// TIA Portal project "station 1 complete twin" (V17)

(* hardware
DEVICE "S7-1500/ET200MP station_1"  S7-1500 station
   slot 0: "Rail_0"  Rack  6ES7 590-1***0-0AA0
   slot 1: "PLC_1"  CPU 1511C-1 PN  6ES7 511-1CK01-0AB0  V2.6
      slot 3: "CPU display_1"  6ES7591-1AA00-0AA0
      slot 32768: "PROFINET interface_1"  X1
         slot 32769: "Port_1"  X1 P1
         slot 32770: "Port_2"  X1 P2
*)

// ===== PLC "PLC_1"  CPU 1511C-1 PN =====

VAR_GLOBAL   // PLC tag table "Default tag table"
   "Tag_1" AT %M0.0 : Bool;
END_VAR

DATA_BLOCK "Station 1"   // DB1
{ S7_Optimized_Access := 'TRUE' }
VERSION : 0.1
   VAR
      Start : Bool;
      Stop : Bool;
      Feed_cylinder : Bool;
      Carriage : Bool;
      Pick_Up_Cylinder : Bool;
      Gripper : Bool;
      System_ON : Bool;
      Workpiece_present : Bool;
      Steps : Int;
      Feed_Cyl_Fully_Extended : Bool;
      Feed_Cyl_Fully_Retracted : Bool;
      Gripper_fully_extended : Bool;
      Gripper_fully_retracted : Bool;
      Carriage_fully_extended : Bool;
      Carriage_fully_retracted : Bool;
   END_VAR
BEGIN
END_DATA_BLOCK

ORGANIZATION_BLOCK "Main"   // OB1, LAD, ProgramCycle
TITLE = "Main Program Sweep (Cycle)"
{ S7_Optimized_Access := 'TRUE' }
VERSION : 0.1
   VAR_INPUT
      Initial_Call : Bool;   // Initial call of this OB
      Remanence : Bool;   // =True, if remanent data are available
   END_VAR
   VAR_TEMP   // added for the SCL form of the ladder/FBD networks
      _w1 : Bool;
   END_VAR
BEGIN

REGION Network 1: Pressing the start button
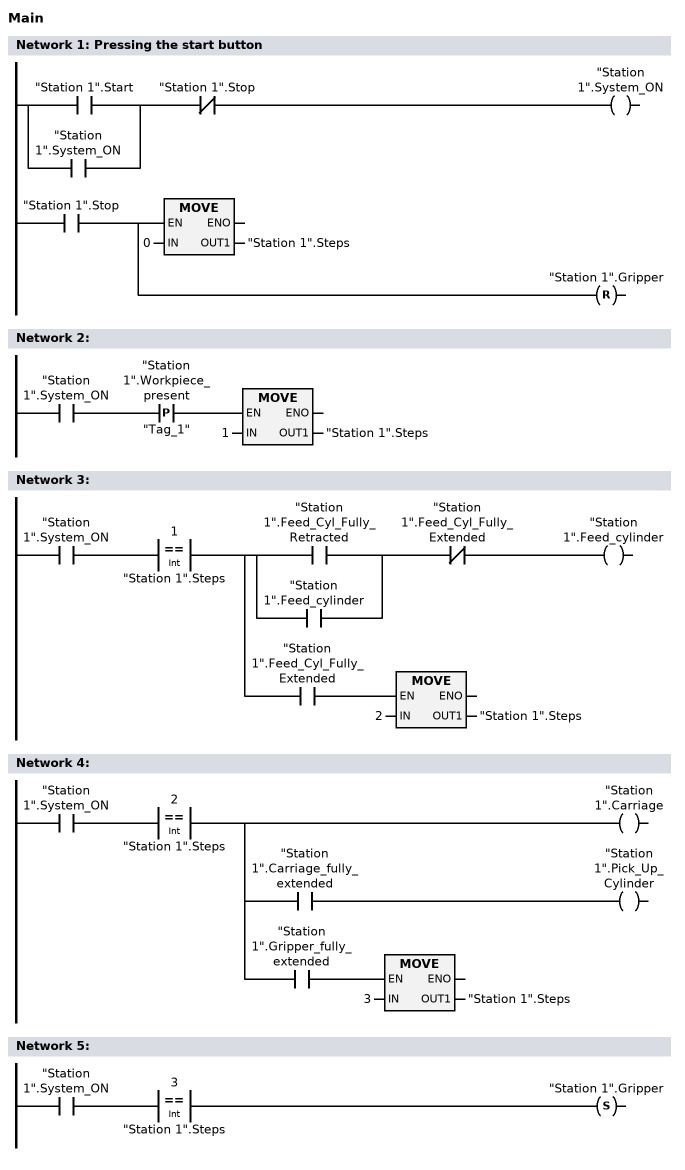
   RUNG wire#powerrail
      Contact( "Station 1".Start )
      wire#w1
      I_Contact( "Station 1".Stop )
      Coil( "Station 1".System_ON )
   END_RUNG
   RUNG wire#powerrail
      Contact( "Station 1".System_ON )
   END_RUNG wire#w1
   RUNG wire#powerrail
      Contact( "Station 1".Stop )
      wire#w2
      Move(in := 0, out1 => "Station 1".Steps)
   END_RUNG
   RUNG wire#w2
      R_Coil( "Station 1".Gripper )
   END_RUNG
   // the same network as SCL:
   "Station 1".System_ON := ("Station 1".Start OR "Station 1".System_ON) AND NOT "Station 1".Stop;
   IF "Station 1".Stop THEN
       "Station 1".Steps := 0;
       "Station 1".Gripper := FALSE;
   END_IF;
END_REGION

REGION Network 2
   RUNG wire#powerrail
      Contact( "Station 1".System_ON )
      P_Contact(operand := "Station 1".Workpiece_present, bit := "Tag_1")
      Move(in := 1, out1 => "Station 1".Steps)
   END_RUNG
   // the same network as SCL:
   #_w1 := "Station 1".System_ON AND "Station 1".Workpiece_present AND NOT "Tag_1";   // rising edge of "Station 1".Workpiece_present
   "Tag_1" := "Station 1".Workpiece_present;
   IF #_w1 THEN "Station 1".Steps := 1; END_IF;
END_REGION

REGION Network 3
   RUNG wire#powerrail
      Contact( "Station 1".System_ON )
      { S7_Templates := "SrcType := Int" } EQ_Contact(in1 := 1, in2 := "Station 1".Steps)
      wire#w1
      Contact( "Station 1".Feed_Cyl_Fully_Retracted )
      wire#w2
      I_Contact( "Station 1".Feed_Cyl_Fully_Extended )
      Coil( "Station 1".Feed_cylinder )
   END_RUNG
   RUNG wire#w1
      Contact( "Station 1".Feed_cylinder )
   END_RUNG wire#w2
   RUNG wire#w1
      Contact( "Station 1".Feed_Cyl_Fully_Extended )
      Move(in := 2, out1 => "Station 1".Steps)
   END_RUNG
   // the same network as SCL:
   #_w1 := "Station 1".System_ON AND (1 = "Station 1".Steps);
   "Station 1".Feed_cylinder := #_w1 AND ("Station 1".Feed_Cyl_Fully_Retracted OR "Station 1".Feed_cylinder) AND NOT "Station 1".Feed_Cyl_Fully_Extended;
   IF #_w1 AND "Station 1".Feed_Cyl_Fully_Extended THEN "Station 1".Steps := 2; END_IF;
END_REGION

REGION Network 4
   RUNG wire#powerrail
      Contact( "Station 1".System_ON )
      { S7_Templates := "SrcType := Int" } EQ_Contact(in1 := 2, in2 := "Station 1".Steps)
      wire#w1
      Coil( "Station 1".Carriage )
   END_RUNG
   RUNG wire#w1
      Contact( "Station 1".Carriage_fully_extended )
      Coil( "Station 1".Pick_Up_Cylinder )
   END_RUNG
   RUNG wire#w1
      Contact( "Station 1".Gripper_fully_extended )
      Move(in := 3, out1 => "Station 1".Steps)
   END_RUNG
   // the same network as SCL:
   "Station 1".Carriage := "Station 1".System_ON AND (2 = "Station 1".Steps);
   "Station 1".Pick_Up_Cylinder := "Station 1".Carriage AND "Station 1".Carriage_fully_extended;
   IF "Station 1".Carriage AND "Station 1".Gripper_fully_extended THEN "Station 1".Steps := 3; END_IF;
END_REGION

REGION Network 5
   RUNG wire#powerrail
      Contact( "Station 1".System_ON )
      { S7_Templates := "SrcType := Int" } EQ_Contact(in1 := 3, in2 := "Station 1".Steps)
      S_Coil( "Station 1".Gripper )
   END_RUNG
   // the same network as SCL:
   IF "Station 1".System_ON AND (3 = "Station 1".Steps) THEN "Station 1".Gripper := TRUE; END_IF;
END_REGION
END_ORGANIZATION_BLOCK